Universal Robots URScript: unalign_for_cover.script

def unalign_for_cover():
  global _hidden_verificationVariable=0
  set_tcp(p[-0.0095,-0.328,0.10573,1.2092,-1.2092,1.2092])
  set_target_payload(10.800000, [-0.001000, -0.053000, 0.068000], [0.081228, 0.081228, 0.081228, 0.000000, 0.000000, 0.000000])
  set_tool_communication(False, 115200, 0, 1, 1.5, 3.5)
  set_tool_output_mode(0)
  set_tool_digital_output_mode(0, 1)
  set_tool_digital_output_mode(1, 1)
  set_tool_voltage(0)
  set_standard_analog_input_domain(0, 1)
  set_standard_analog_input_domain(1, 1)
  set_tool_analog_input_domain(0, 1)
  set_tool_analog_input_domain(1, 1)
  set_analog_outputdomain(0, 0)
  set_analog_outputdomain(1, 0)
  set_input_actions_to_default()
  set_gravity([0.0, 0.0, 9.82])
  set_safety_mode_transition_hardness(1)
  global robot_number=2
  global Point_1=p[0.0,0.0,0.0,0.0,0.0,0.0]
  global Point_2=p[0.0,0.0,0.0,0.0,0.0,0.0]
  # begin: URCap Installation Node
  #   Source: UR Connect, 1.13.79, Universal Robots
  #   Type: UR Connect
  myurRPC = rpc_factory("xmlrpc","http://127.0.0.1:40474")
  # end: URCap Installation Node
  # begin: URCap Installation Node
  #   Source: MachineLogic for Universal Robots, 3.1.7, Vention Inc.
  #   Type: MachineLogic for Universal Robots
  def waitForResponse(expected_response_vention, cname_vention):
  response_vention = socket_read_string(cname_vention,timeout=15)
  while response_vention != expected_response_vention:
  sleep(0.01)
  response_vention = socket_read_string(cname_vention,timeout=15)
  end
  sleep(0.01)
  sync()
  end
  def sendString(string_vention, expected_response_vention, cname_vention):
  socket_send_string(str_cat(string_vention,";"), cname_vention)
  response_vention = socket_read_string(cname_vention,timeout=15)
  if(response_vention == "nAck"):
  popup("nAck received")
  end
  while response_vention != expected_response_vention:
  sleep(0.01)
  response_vention = socket_read_string(cname_vention,timeout=15)
  if(response_vention == "nAck"):
  popup("nAck received")
  end
  end
  sleep(0.01)
  sync()
  end
  def sendStringNAck(string_vention, expected_response_vention, cname_vention):
  socket_send_string(str_cat(string_vention,";"), cname_vention)
  response_vention = socket_read_string(cname_vention,timeout=15)
  if(response_vention == "nAck"):
  popup("nAck received")
  end
  while(response_vention != expected_response_vention and response_vention != "nAck"):
  sleep(0.01)
  response_vention = socket_read_string(cname_vention,timeout=15)
  if(response_vention == "nAck"):
  popup("nAck received",blocking=True)
  end
  end
  sleep(0.01)
  sync()
  end
  def sendStringWithTimeout(string_vention, expected_response_vention, cname_vention):
  socket_send_string(str_cat(string_vention,";"), cname_vention)
  response_vention = socket_read_string(cname_vention,timeout=10)
  if(response_vention == "nAck"):
  popup("nAck received"+string_vention)
  end
  sleep(0.01)
  sync()
  end
  def pollString(string_vention, expected_response_vention, cname_vention):
  socket_send_string(str_cat(string_vention,";"), cname_vention)
  response_vention = socket_read_string(cname_vention,timeout=15)
  if(response_vention == "nAck"):
  popup("nAck received")
  end
  while response_vention != expected_response_vention:
  sleep(1)
  socket_send_string(str_cat(string_vention,";"), cname_vention)
  response_vention = socket_read_string(cname_vention,timeout=15)
  if(response_vention == "nAck"):
  popup("nAck received")
  end
  end
  sleep(0.01)
  sync()
  end
  def sendVariable(var_vention, data_vention, expected_response_vention, cname_vention):
  socket_set_var(var_vention, data_vention, cname_vention)
  response_vention = socket_read_string(cname_vention,timeout=15)
  if(response_vention == "nAck"):
  popup("nAck received")
  end
  while response_vention != expected_response_vention:
  sleep(0.01)
  response_vention = socket_read_string(cname_vention,timeout=15)
  if(response_vention == "nAck"):
  popup("nAck received")
  end
  end
  sleep(0.01)
  sync()
  end
  def intToString(integer_vention,cname_vention):
  stringFix=""
  multiplier_vention123=1
  if integer_vention<0:
  stringFix="-"
  multiplier_vention123=-1
  end
  socket_set_var("GetString",integer_vention*multiplier_vention123,cname_vention)
  string_vention=""
  while string_vention=="":
  sleep(0.01)
  string_vention=socket_read_string(cname_vention,timeout=15)
  end
  sleep(0.01)
  sync()
  string_vention=stringFix+string_vention
  return string_vention
  end
  string_vention=""
  isVentionMovementBusy = False
  isVentionParallelMovementSendingScript = False
  ventionThreadHandle = 1
  isVentionMovementBusyMachineMotion1 = False
  isVentionParallelMovementSendingScriptMachineMotion1 = False
  socket_vention = socket_open("192.168.3.52", 9999, "MachineMotion1")
  if socket_vention==False:
  popup("Check configuration, can't connect to MachineMotion")
  end
  waitForResponse("MachineMotion connection established", "MachineMotion1")
  sendString("isReady", "MachineMotion isReady = true", "MachineMotion1")
  sendStringWithTimeout("setURCapVersion2", "setURCapVersion loaded", "MachineMotion1")
  sendString("SET speed_v2 1000000", "Ack", "MachineMotion1")
  sendString("SET acceleration_v2 100000", "Ack", "MachineMotion1")
  sendString("SET de_axis_1_microsteps_config 8", "Ack", "MachineMotion1")
  sendString("SET de_axis_1_mechanical_gain_config_v2 150000.0", "Ack", "MachineMotion1")
  sendString("SET de_axis_1_direction_config 1", "Ack", "MachineMotion1")
  sendString("SET de_axis_1_type_config Custom Actuator ", "Ack", "MachineMotion1")
  sendString("de_axis_1_config_exec", "Ack", "MachineMotion1")
  # end: URCap Installation Node
  # begin: URCap Installation Node
  #   Source: WireTank Serial, 4.9.0, WireTank, LLC
  #   Type: WireTank Serial
  WTSerialBridge = rpc_factory("xmlrpc","http://127.0.0.1:40511/RPC2")
  # end: URCap Installation Node
  step_count_6066afa7_6d3e_40c2_b283_208ec4fe33a3 = 0.0
  thread Step_Counter_Thread_5cae079c_b6a8_4d9c_956a_44e16054eccd():
    while (True):
      step_count_6066afa7_6d3e_40c2_b283_208ec4fe33a3 = step_count_6066afa7_6d3e_40c2_b283_208ec4fe33a3 + 1.0
      sync()
    end
  end
  run Step_Counter_Thread_5cae079c_b6a8_4d9c_956a_44e16054eccd()
  def calculate_point_to_move_towards(feature, direction, position_distance):
    local posDir=[direction[0], direction[1], direction[2]]
    if (norm(posDir) < 1e-6):
      return get_target_waypoint()
    end
    local direction_vector_normalized=normalize(posDir)
    local displacement_pose=p[direction_vector_normalized[0] * position_distance,direction_vector_normalized[1] * position_distance,direction_vector_normalized[2] * position_distance,0,0,0]
    local wanted_displacement_in_base_frame=pose_sub(pose_trans(feature, displacement_pose), feature)
    return pose_add(get_target_waypoint(), wanted_displacement_in_base_frame)
  end
  global Waypoint_9_p=p[-.242109381762, .328859740510, .325759000406, -1.405332652358, 1.226734092173, -1.029352124345]
  global Waypoint_9_q=[-3.630085628802167, -1.8749691927959926, -2.036734414610116, -2.3725978513806703, -3.7650640868214893, 1.3954688983392125]
  global Waypoint_10_p=p[-.240919897414, .326606982418, .327046253747, -.783499228114, 1.948636770247, -1.629561181456]
  global Waypoint_10_q=[-4.098476127203824, -1.8560160055412283, -2.0602626111701134, -2.371189229470515, -3.2917242638401625, 1.38870966600456]
  $ 2 "Robot Program"
  $ 25 "actualprogram"
  $ 26 "MoveL"
  $ 27 "Direction: Base X+"
  global move_thread_flag_27=0
  thread move_thread_27():
    enter_critical
    move_thread_flag_27 = 1
    local towardsPos=calculate_point_to_move_towards(p[0.0,0.0,0.0,0.0,0.0,0.0], [1.0,0.0,0.0], 0.15)
    movel(towardsPos, a=1.2, v=0.25)
    move_thread_flag_27 = 2
    exit_critical
  end
  move_thread_flag_27 = 0
  move_thread_han_27 = run move_thread_27()
  while (True):
    sleep(1.0E-10)
    if (move_thread_flag_27 > 1):
      join move_thread_han_27
      $ 28 "Until (distance)"
      break
    end
    sync()
  end
  $ 29 "MoveL"
  $ 30 "Direction: Base Z+"
  global move_thread_flag_30=0
  thread move_thread_30():
    enter_critical
    move_thread_flag_30 = 1
    local towardsPos=calculate_point_to_move_towards(p[0.0,0.0,0.0,0.0,0.0,0.0], [0.0,0.0,1.0], 0.2)
    movel(towardsPos, a=1.2, v=0.25)
    move_thread_flag_30 = 2
    exit_critical
  end
  move_thread_flag_30 = 0
  move_thread_han_30 = run move_thread_30()
  while (True):
    sleep(1.0E-10)
    if (move_thread_flag_30 > 1):
      join move_thread_han_30
      $ 31 "Until (distance)"
      break
    end
    sync()
  end
  $ 32 "MoveJ"
  $ 33 "Waypoint_9" "breakAfter"
  movej(get_inverse_kin(Waypoint_9_p, qnear=Waypoint_9_q), a=1.3962634015954636, v=1.0471975511965976)
  $ 34 "Waypoint_10" "breakAfter"
  movej(get_inverse_kin(Waypoint_10_p, qnear=Waypoint_10_q), a=1.3962634015954636, v=1.0471975511965976)
  $ 35 "Home"
  movej([-3.266929759358355, -1.2139462677784536, 1.5878387874396154, 1.1069165929565088, -0.0023738326664366483, -1.7891447305770605], a=1.3962634015954636, v=1.0471975511965976)
  # begin: URCap Program Node
  #   Source: MachineLogic for Universal Robots, 3.1.7, Vention Inc.
  #   Type: MachineLogic for Universal Robots
  $ 36 "MachineLogic Homing"
  while isVentionMovementBusyMachineMotion1==True:
  sleep(0.05)
  end
  if(isVentionMovementBusyMachineMotion1 == False):
  isVentionMovementBusyMachineMotion1 = True
  socket_send_string("estop/status;", "MachineMotion1")
  temp_estop_var_vention = socket_read_string("MachineMotion1",timeout=15)
  while(temp_estop_var_vention=="estop/status true"):
  if temp_estop_var_vention=="estop/status true":
  sendStringWithTimeout("estop/systemreset/request","Ack estop/systemreset/request;","MachineMotion1")
  end
  socket_send_string("estop/status;", "MachineMotion1")
  temp_estop_var_vention = socket_read_string("MachineMotion1",timeout=15)
  if temp_estop_var_vention=="estop/status true":
  popup("MachineMotion in estop, make sure you have all emergency modules released manually. If you continue the system will try to reset MachineMotion automatically.",blocking=True)
  end
  end
  else:
  popup("resource is being used already: MachineMotion1")
  halt
  end
  isVentionMovementBusyMachineMotion1 = True
  sendString("im_home_axis_1", "MachineMotion im_home_axis_1 = completed", "MachineMotion1")
  isVentionMovementBusyMachineMotion1 = False
  sendString("SET im_set_encoder_pos_aux_1 0.000", "Ack", "MachineMotion1")
  isVentionMovementBusyMachineMotion1 = False
  sleep(0.03)
  # end: URCap Program Node
end
